{attribute 'linkalways'} 
{attribute 'no_explicit_call' := 'This FB is a CLASS and must be accessed using methods or properties'}
{attribute 'enable_dynamic_creation'}
FUNCTION_BLOCK Node_F_VN_FillCircle EXTENDS VisionNode
VAR
    nCenterX : _UDINT(0);
    nCenterY : _UDINT(0);
    nRadius : _UDINT(0);
    ipDestImage : _ITcVnImage;
    aColor : _TcVnVector4_LREAL;
    hrPrev : _HRESULT(S_OK);
	hresult : _HRESULT(S_OK);
END_VAR

METHOD PUBLIC  Clone : I_Node
VAR
	pNode : POINTER TO Node_F_VN_FillCircle;
END_VAR
pNode := __NEW(Node_F_VN_FillCircle);
Clone := pNode^;
END_METHOD

METHOD FB_init : BOOL
VAR_INPUT
	bInitRetains : BOOL; // if TRUE, the retain variables are initialized (warm start / cold start)
	bInCopyCode : BOOL;  // if TRUE, the instance afterwards gets moved into the copy code (online change)
END_VAR
AddInput('nCenterX', nCenterX);
AddInput('nCenterY', nCenterY);
AddInput('nRadius', nRadius);
AddInput('ipDestImage', ipDestImage);
AddInput('aColor', aColor);
AddInput('hrPrev', hrPrev);
AddOutput('ipDestImage', ipDestImage);
AddOutput('hresult',hresult);
END_METHOD

METHOD PROTECTED  OnExecute : HRESULT
hresult.Value := F_VN_FillCircle(
    nCenterX := nCenterX.Value,
    nCenterY := nCenterY.Value,
    nRadius := nRadius.Value,
	ipDestImage := ipDestImage.Value,
    aColor := aColor.Value,
	hrPrev:= hrPrev.Value);
END_METHOD

METHOD PUBLIC PreExecutionCheck
VAR_INPUT
	Check : I_PreExecutionChecks;
END_VAR
Check.IsTrue(ipDestImage.IsValid, 'ipDestImage must contain an image');
END_METHOD

END_FUNCTION_BLOCK

(* stored: Version 1.1.0.1, ProductVersion 3.1.4024.13
   POU Node_F_VN_FillCircle: Id {f84a3d8d-823f-0b79-3547-3f60c4244b2f}, SpecialFunc None
   Folder Constructor: Id {e7f343de-c0b9-0389-2dd6-9b638e8ba6e0}
   Method Clone: Id {1f0bdde4-09e3-0a52-2009-e5a46e616343}
   Method FB_init: Id {78e77074-07d3-0839-2fac-da12d29582c2}
   Method OnExecute: Id {64ac9e55-162c-0c2d-094d-b1f7a8f288b6}
   Method PreExecutionCheck: Id {2e38ea4f-ed64-062b-32bd-6d0ac8f1e5f5} *)
